FUNCTION_BLOCK Grade_Comandos (* Composite Function Block Type *)
  (* Standard: 61499-2 *)
  (* Version 0.0, 2/24/2026, template *)
  PACKAGE Hidryco.HidrycoLib;
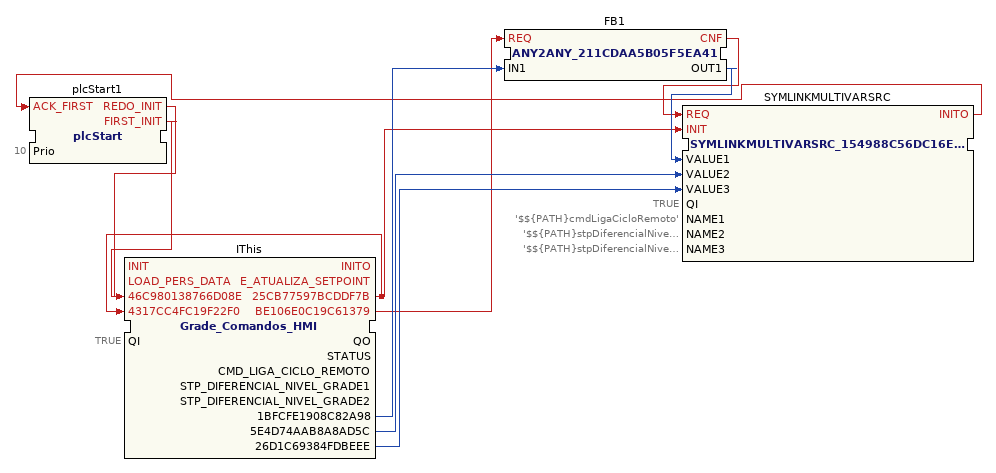
  FBS
    IThis : Grade_Comandos_HMI(QI := TRUE);
    plcStart1 : plcStart(Prio := 10);
    FB1 : ANY2ANY_211CDAA5B05F5EA41; {SET_ATTRIBUTE(Configuration.GenericFBType.InterfaceParams, Runtime.Standard#CNT:=1;IN${CNT$}:BOOL;OUT${CNT$}:INT)}
    SYMLINKMULTIVARSRC : SYMLINKMULTIVARSRC_154988C56DC16E7CE(QI := TRUE, NAME1 := '$${PATH}cmdLigaCicloRemoto', NAME2 := '$${PATH}stpDiferencialNivelGrade1', NAME3 := '$${PATH}stpDiferencialNivelGrade2'); {SET_ATTRIBUTE(Configuration.GenericFBType.InterfaceParams, Runtime.System#I:=3;VALUE${I$}:INT,INT,INT)}
  END_FBS
  EVENT_CONNECTIONS
    FB1.CNF TO SYMLINKMULTIVARSRC.REQ;
    plcStart1.REDO_INIT TO IThis.46C980138766D08E;
    plcStart1.FIRST_INIT TO IThis.46C980138766D08E;
    IThis.25CB77597BCDDF7B TO IThis.4317CC4FC19F22F0;
    IThis.25CB77597BCDDF7B TO SYMLINKMULTIVARSRC.INIT;
    IThis.BE106E0C19C61379 TO FB1.REQ;
    SYMLINKMULTIVARSRC.INITO TO plcStart1.ACK_FIRST;
  END_CONNECTIONS
  DATA_CONNECTIONS
    FB1.OUT1 TO SYMLINKMULTIVARSRC.VALUE1;
    IThis.1BFCFE1908C82A98 TO FB1.IN1;
    IThis.5E4D74AAB8A8AD5C TO SYMLINKMULTIVARSRC.VALUE2;
    IThis.26D1C69384FDBEEE TO SYMLINKMULTIVARSRC.VALUE3;
  END_CONNECTIONS
END_FUNCTION_BLOCK
